FUNCTION_BLOCK UT_AuxiliaryInputMapping (* Service Interface Function Block Type *)
  (* Standard: ISO 11783-6; Classification: Button – ISO 11783-6 – B.7; Function: All Inputs; Type: UT according to ISO 11783-6 *)
  (* Version 1.0, 2018-12-05, Jose Cabral *)
  (* Version 1.0, 2022-08-04, Franz Höpfinger, Unknown *)
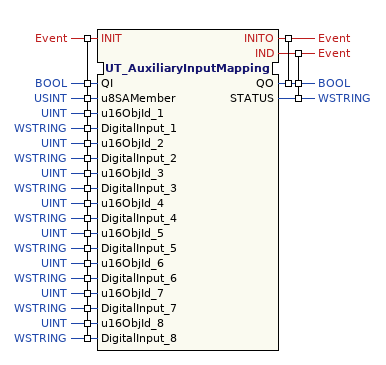
  EVENT_INPUT
    INIT WITH QI, u8SAMember, u16ObjId_1, DigitalInput_1, u16ObjId_2, DigitalInput_2, u16ObjId_3, DigitalInput_3, u16ObjId_4, DigitalInput_4, u16ObjId_5, DigitalInput_5, u16ObjId_6, DigitalInput_6, u16ObjId_7, DigitalInput_7, u16ObjId_8, DigitalInput_8; (* Service Initialization *)
  END_EVENT
  EVENT_OUTPUT
    INITO WITH QO; (* Initialization Confirm *)
    IND WITH QO, STATUS; (* Indication from Resource *)
  END_EVENT
  VAR_INPUT
    QI : BOOL; (* Event Input Qualifier *)
    u8SAMember : USINT := 255; (* Dummy !, set to 255 if in doubt. 0 deactivates FB. *)
    u16ObjId_1 : UINT := 31000; (* Object ID of Input 1 *)
    DigitalInput_1 : WSTRING := "AuxInput_31000"; (* Identifier for Input 1 *)
    u16ObjId_2 : UINT := 31001; (* Object ID of Input 2 *)
    DigitalInput_2 : WSTRING := "AuxInput_31001"; (* Identifier for Input 2 *)
    u16ObjId_3 : UINT := 31002; (* Object ID of Input 3 *)
    DigitalInput_3 : WSTRING := "AuxInput_31002"; (* Identifier for Input 3 *)
    u16ObjId_4 : UINT := 31003; (* Object ID of Input 4 *)
    DigitalInput_4 : WSTRING := "AuxInput_31003"; (* Identifier for Input 4 *)
    u16ObjId_5 : UINT := 31004; (* Object ID of Input 5 *)
    DigitalInput_5 : WSTRING := "AuxInput_31004"; (* Identifier for Input 5 *)
    u16ObjId_6 : UINT := 31005; (* Object ID of Input 6 *)
    DigitalInput_6 : WSTRING := "AuxInput_31005"; (* Identifier for Input 6 *)
    u16ObjId_7 : UINT := 31006; (* Object ID of Input 7 *)
    DigitalInput_7 : WSTRING := "AuxInput_31006"; (* Identifier for Input 7 *)
    u16ObjId_8 : UINT := 31007; (* Object ID of Input 8 *)
    DigitalInput_8 : WSTRING := "AuxInput_31007"; (* Identifier for Input 8 *)
  END_VAR
  VAR_OUTPUT
    QO : BOOL; (* Event Output Qualifier *)
    STATUS : WSTRING; (* Service Status *)
  END_VAR
END_FUNCTION_BLOCK
